{attribute 'linkalways'} 
{attribute 'no_explicit_call' := 'This FB is a CLASS and must be accessed using methods or properties'}
{attribute 'enable_dynamic_creation'}
FUNCTION_BLOCK JsonDeserializer EXTENDS Disposable IMPLEMENTS I_Deserializer
VAR
	jsonParser : JsonDomParser;
	root : SJsonValue;
	garbageCollector : DeserializerGarbageCollector;
	nullNode : JsonDeserializerNullNode;
	rootNode : I_Deserializer := nullNode;
END_VAR

METHOD PUBLIC Clone : I_Deserializer
VAR
	pClone : POINTER TO JsonDeserializer;
	jsonSize : UDINT;
	pJsonString : POINTER TO STRING;
END_VAR
pClone := __NEW(JsonDeserializer);
Clone := pClone^;

jsonSize := jsonParser.GetDocumentLength();

IF jsonSize = 0 THEN
	// no further cloning to do. 
	RETURN;
END_IF

pJsonString := __NEW(BYTE, jsonSize);

IF jsonParser.CopyDocument(pJsonString^, jsonSize) = 0 THEN
	__DELETE(pJsonString);
	RETURN;
END_IF

pClone^.TryLoad(pJsonString^);
__DELETE(pJsonString);
END_METHOD

METHOD PROTECTED CreateDeserializer : I_Deserializer
VAR_INPUT
	DeserializerRoot : SJsonValue;
END_VAR
VAR 
	pNode : POINTER TO JsonDeserializerNode;
END_VAR
pNode := __NEW(JsonDeserializerNode(ParentJsonDomParser := jsonParser, NodeRoot := DeserializerRoot, ParentGarbageCollector := garbageCollector, ParentNullDeserializer := nullNode));
CreateDeserializer := pNode^;
END_METHOD

METHOD FB_exit : BOOL
VAR_INPUT
	bInCopyCode : BOOL; // if TRUE, the exit method is called for exiting an instance that is copied afterwards (online change).
END_VAR
IF bInCopyCode THEN
	RETURN;
END_IF

Reset();
END_METHOD

METHOD GetArray : I_Deserializer
VAR_INPUT
END_VAR
GetArray := rootNode.GetArray();
END_METHOD

METHOD GetElementByIndex : I_Deserializer
VAR_INPUT
	Index : UDINT;
END_VAR
GetElementByIndex := rootNode.GetElementByIndex(Index);
END_METHOD

METHOD GetKey : I_Deserializer
VAR_INPUT
	Key : T_MAXSTRING;
END_VAR
GetKey := rootNode.GetKey(Key);
END_METHOD

METHOD GetKeyArray : I_Deserializer
VAR_INPUT
	Key : T_MAXSTRING;
END_VAR
GetKeyArray := rootNode.GetKeyArray(Key);
END_METHOD

METHOD PUBLIC Reset
VAR_INPUT
END_VAR
jsonParser.NewDocument();
garbageCollector.Execute();
root := 0;
rootNode := nullNode;
END_METHOD

METHOD TryGetBase64 : BOOL
VAR_INPUT
	pBytes : POINTER TO BYTE;
	nBytes : DINT;
END_VAR
TryGetBase64 := rootNode.TryGetBase64(pBytes, nBytes);
END_METHOD

METHOD TryGetBool : BOOL
VAR_INPUT
	Destination : REFERENCE TO BOOL;
END_VAR
TryGetBool := rootNode.TryGetBool(Destination);
END_METHOD

METHOD TryGetByte : BOOL
VAR_INPUT
	Destination : REFERENCE TO BYTE;
END_VAR
TryGetByte := rootNode.TryGetByte(Destination);
END_METHOD

METHOD TryGetDateTime : BOOL
VAR_INPUT
	Destination : REFERENCE TO DATE_AND_TIME;
END_VAR
TryGetDateTime := rootNode.TryGetDateTime(Destination);
END_METHOD

METHOD TryGetDcTime : BOOL
VAR_INPUT
	Destination : REFERENCE TO DCTIME;
END_VAR
TryGetDcTime := rootNode.TryGetDcTime(Destination);
END_METHOD

METHOD TryGetDint : BOOL
VAR_INPUT
	Destination : REFERENCE TO DINT;
END_VAR
TryGetDint := rootNode.TryGetDint(Destination);
END_METHOD

METHOD TryGetDword : BOOL
VAR_INPUT
	Destination : REFERENCE TO DWORD;
END_VAR
TryGetDword := rootNode.TryGetDword(Destination);
END_METHOD

METHOD TryGetFileTime : BOOL
VAR_INPUT
	Destination : REFERENCE TO FILETIME;
END_VAR
TryGetFileTime := rootNode.TryGetFileTime(Destination);
END_METHOD

METHOD TryGetHexAsBytes : BOOL
VAR_INPUT
	pBytes : POINTER TO BYTE;
	nBytes : DINT;
END_VAR
TryGetHexAsBytes := rootNode.TryGetHexAsBytes(pBytes, nBytes);
END_METHOD

METHOD TryGetInt : BOOL
VAR_INPUT
	Destination : REFERENCE TO INT;
END_VAR
TryGetInt := rootNode.TryGetInt(Destination);
END_METHOD

METHOD TryGetKeyBase64 : BOOL
VAR_INPUT
	Key : T_MAXSTRING;
	pBytes : POINTER TO BYTE;
	nBytes : DINT;
END_VAR
TryGetKeyBase64 := rootNode.TryGetKeyBase64(Key, pBytes, nBytes);
END_METHOD

METHOD TryGetKeyBool : BOOL
VAR_INPUT
	Key : T_MAXSTRING;
	Destination : REFERENCE TO BOOL;
END_VAR
TryGetKeyBool := rootNode.TryGetKeyBool(Key, Destination);
END_METHOD

METHOD TryGetKeyByte : BOOL
VAR_INPUT
	Key : T_MAXSTRING;
	Destination : REFERENCE TO BYTE;
END_VAR
TryGetKeyByte := rootNode.TryGetKeyByte(Key, Destination);
END_METHOD

METHOD TryGetKeyDateTime : BOOL
VAR_INPUT
	Key : T_MAXSTRING;
	Destination : REFERENCE TO DATE_AND_TIME;
END_VAR
TryGetKeyDateTime := rootNode.TryGetKeyDateTime(Key, Destination);
END_METHOD

METHOD TryGetKeyDcTime : BOOL
VAR_INPUT
	Key : T_MAXSTRING;
	Destination : REFERENCE TO DCTIME;
END_VAR
TryGetKeyDcTime := rootNode.TryGetKeyDcTime(Key, Destination);
END_METHOD

METHOD TryGetKeyDint : BOOL
VAR_INPUT
	Key : T_MAXSTRING;
	Destination : REFERENCE TO DINT;
END_VAR
TryGetKeyDint := rootNode.TryGetKeyDint(Key, Destination);
END_METHOD

METHOD TryGetKeyDword : BOOL
VAR_INPUT
	Key : T_MAXSTRING;
	Destination : REFERENCE TO DWORD;
END_VAR
TryGetKeyDword := rootNode.TryGetKeyDword(Key, Destination);
END_METHOD

METHOD TryGetKeyFileTime : BOOL
VAR_INPUT
	Key : T_MAXSTRING;
	Destination : REFERENCE TO FILETIME;
END_VAR
TryGetKeyFileTime := rootNode.TryGetKeyFileTime(Key, Destination);
END_METHOD

METHOD TryGetKeyHexAsBytes : BOOL
VAR_INPUT
	Key : T_MAXSTRING;
	pBytes : POINTER TO BYTE;
	nBytes : DINT;
END_VAR
TryGetKeyHexAsBytes := rootNode.TryGetKeyHexAsBytes(Key, pBytes, nBytes);
END_METHOD

METHOD TryGetKeyInt : BOOL
VAR_INPUT
	Key : T_MAXSTRING;
	Destination : REFERENCE TO INT;
END_VAR
TryGetKeyInt := rootNode.TryGetKeyInt(Key, Destination);
END_METHOD

METHOD TryGetKeyLint : BOOL
VAR_INPUT
	Key : T_MAXSTRING;
	Destination : REFERENCE TO LINT;
END_VAR
TryGetKeyLint := rootNode.TryGetKeyLint(Key, Destination);
END_METHOD

METHOD TryGetKeyLreal : BOOL
VAR_INPUT
	Key : T_MAXSTRING;
	Destination : REFERENCE TO LREAL;
END_VAR
TryGetKeyLreal := rootNode.TryGetKeyLreal(Key, Destination);
END_METHOD

METHOD TryGetKeyLtime : BOOL
VAR_INPUT
	Key : T_MAXSTRING;
	Destination : REFERENCE TO LTIME;
END_VAR
TryGetKeyLtime := rootNode.TryGetKeyLtime(Key, Destination);
END_METHOD

METHOD TryGetKeyLword : BOOL
VAR_INPUT
	Key : T_MAXSTRING;
	Destination : REFERENCE TO LWORD;
END_VAR
TryGetKeyLword := rootNode.TryGetKeyLword(Key, Destination);
END_METHOD

METHOD TryGetKeyObject : BOOL
VAR_INPUT
	Key : T_MAXSTRING;
	Object : I_Deserializable;
END_VAR
TryGetKeyObject := rootNode.TryGetKeyObject(Key,Object);
END_METHOD

METHOD TryGetKeyReal : BOOL
VAR_INPUT
	Key : T_MAXSTRING;
	Destination : REFERENCE TO REAL;
END_VAR
TryGetKeyReal := rootNode.TryGetKeyReal(Key, Destination);
END_METHOD

METHOD TryGetKeySint : BOOL
VAR_INPUT
	Key : T_MAXSTRING;
	Destination : REFERENCE TO SINT;
END_VAR
TryGetKeySint := rootNode.TryGetKeySint(Key, Destination);
END_METHOD

METHOD TryGetKeyString : BOOL
VAR_INPUT
	Key : T_MAXSTRING;
	Destination : REFERENCE TO STRING;
END_VAR
TryGetKeyString := rootNode.TryGetKeyString(Key, Destination);
END_METHOD

METHOD TryGetKeyTime : BOOL
VAR_INPUT
	Key : T_MAXSTRING;
	Destination : REFERENCE TO TIME;
END_VAR
TryGetKeyTime := rootNode.TryGetKeyTime(Key, Destination);
END_METHOD

METHOD TryGetKeyTod : BOOL
VAR_INPUT
	Key : T_MAXSTRING;
	Destination : REFERENCE TO TOD;
END_VAR
TryGetKeyTod := rootNode.TryGetKeyTod(Key, Destination);
END_METHOD

METHOD TryGetKeyUdint : BOOL
VAR_INPUT
	Key : T_MAXSTRING;
	Destination : REFERENCE TO UDINT;
END_VAR
TryGetKeyUdint := rootNode.TryGetKeyUdint(Key, Destination);
END_METHOD

METHOD TryGetKeyUint : BOOL
VAR_INPUT
	Key : T_MAXSTRING;
	Destination : REFERENCE TO UINT;
END_VAR
TryGetKeyUint := rootNode.TryGetKeyUint(Key, Destination);
END_METHOD

METHOD TryGetKeyUlint : BOOL
VAR_INPUT
	Key : T_MAXSTRING;
	Destination : REFERENCE TO ULINT;
END_VAR
TryGetKeyUlint := rootNode.TryGetKeyUlint(Key, Destination);
END_METHOD

METHOD TryGetKeyUsint : BOOL
VAR_INPUT
	Key : T_MAXSTRING;
	Destination : REFERENCE TO USINT;
END_VAR
TryGetKeyUsint := rootNode.TryGetKeyUsint(Key, Destination);
END_METHOD

METHOD TryGetKeyWord : BOOL
VAR_INPUT
	Key : T_MAXSTRING;
	Destination : REFERENCE TO WORD;
END_VAR
TryGetKeyWord := rootNode.TryGetKeyWord(Key, Destination);
END_METHOD

METHOD TryGetLint : BOOL
VAR_INPUT
	Destination : REFERENCE TO LINT;
END_VAR
TryGetLint := rootNode.TryGetLint(Destination);
END_METHOD

METHOD TryGetLreal : BOOL
VAR_INPUT
	Destination : REFERENCE TO LREAL;
END_VAR
TryGetLreal := rootNode.TryGetLreal(Destination);
END_METHOD

METHOD TryGetLtime : BOOL
VAR_INPUT
	Destination : REFERENCE TO LTIME;
END_VAR
TryGetLtime := rootNode.TryGetLtime(Destination);
END_METHOD

METHOD TryGetLword : BOOL
VAR_INPUT
	Destination : REFERENCE TO LWORD;
END_VAR
TryGetLword := rootNode.TryGetLword(Destination);
END_METHOD

METHOD TryGetObject : BOOL
VAR_INPUT
	Object : I_Deserializable;
END_VAR
TryGetObject := rootNode.TryGetObject(Object);
END_METHOD

METHOD TryGetReal : BOOL
VAR_INPUT
	Destination : REFERENCE TO REAL;
END_VAR
TryGetReal := rootNode.TryGetReal(Destination);
END_METHOD

METHOD TryGetSint : BOOL
VAR_INPUT
	Destination : REFERENCE TO SINT;
END_VAR
TryGetSint := rootNode.TryGetSint(Destination);
END_METHOD

METHOD TryGetString : BOOL
VAR_INPUT
	Destination : REFERENCE TO STRING;
END_VAR
TryGetString := rootNode.TryGetString(Destination);
END_METHOD

METHOD TryGetTime : BOOL
VAR_INPUT
	Destination : REFERENCE TO TIME;
END_VAR
TryGetTime := rootNode.TryGetTime(Destination);
END_METHOD

METHOD TryGetTod : BOOL
VAR_INPUT
	Destination : REFERENCE TO TOD;
END_VAR
TryGetTod := rootNode.TryGetTod(Destination);
END_METHOD

METHOD TryGetUdint : BOOL
VAR_INPUT
	Destination : REFERENCE TO UDINT;
END_VAR
TryGetUdint := rootNode.TryGetUdint(Destination);
END_METHOD

METHOD TryGetUint : BOOL
VAR_INPUT
	Destination : REFERENCE TO UINT;
END_VAR
TryGetUint := rootNode.TryGetUint(Destination);
END_METHOD

METHOD TryGetUlint : BOOL
VAR_INPUT
	Destination : REFERENCE TO ULINT;
END_VAR
TryGetUlint := rootNode.TryGetUlint(Destination);
END_METHOD

METHOD TryGetUsint : BOOL
VAR_INPUT
	Destination : REFERENCE TO USINT;
END_VAR
TryGetUsint := rootNode.TryGetUsint(Destination);
END_METHOD

METHOD TryGetWord : BOOL
VAR_INPUT
	Destination : REFERENCE TO WORD;
END_VAR
TryGetWord := rootNode.TryGetWord(Destination);
END_METHOD

METHOD PUBLIC TryLoad : BOOL
VAR_INPUT
	SerializedData : REFERENCE TO STRING;;
END_VAR
Reset();

root := jsonParser.ParseDocument(SerializedData);
IF root = 0 THEN
	RETURN;
END_IF

rootNode := CreateDeserializer(root);
TryLoad := TRUE;
END_METHOD

END_FUNCTION_BLOCK

(* stored: Version 1.1.0.1, ProductVersion 3.1.4024.12
   POU JsonDeserializer: Id {a90a43d9-ea62-48ae-9b56-2bc4217891a9}, SpecialFunc None
   Folder Destructor: Id {bf822394-22a2-42d6-8812-78eace02343d}
   Folder Protected: Id {01c55fae-a423-471f-adbb-267168f4fce0}
   Method Clone: Id {f09ba639-152e-42ab-83f4-0db39532c374}
   Method CreateDeserializer: Id {6e178c51-cb69-40a4-96bf-b38252df7bdc}
   Method FB_exit: Id {d9f286cf-0a82-45b5-9661-1cb5706a832d}
   Method GetArray: Id {a8b524f2-5f76-4824-97b5-f83f0e1611cd}
   Method GetElementByIndex: Id {adfb94ab-88ff-476c-a549-f0880b6a7e45}
   Method GetKey: Id {0f1075b2-7f5b-4f71-8323-87a91a30b569}
   Method GetKeyArray: Id {64ed3b17-47ab-402e-a2fe-0b75f40cb73a}
   Method Reset: Id {ff410b24-6bd3-4b0b-b181-8baf610127fb}
   Method TryGetBase64: Id {fe295ea1-6385-4c90-8c1e-0130d0abea78}
   Method TryGetBool: Id {6ec60297-fc78-4e42-8c9b-b797b172a63d}
   Method TryGetByte: Id {7f56b251-eee0-4e1f-94af-df45fa90da48}
   Method TryGetDateTime: Id {0eefca34-6e86-480c-bd80-cca9f9d6217f}
   Method TryGetDcTime: Id {822c1511-2a5b-4b36-a7ac-0e7bb0382e3f}
   Method TryGetDint: Id {72d1a2f6-6d1c-43bc-8260-7a62f2ef0180}
   Method TryGetDword: Id {92993be7-2fb3-49bb-aa8c-994491f8b23c}
   Method TryGetFileTime: Id {6f985b02-908a-4e9a-8047-f818f837fe22}
   Method TryGetHexAsBytes: Id {57725d6f-7769-44f1-b87a-65ec295b3672}
   Method TryGetInt: Id {2fdf166b-5700-40ee-b8b0-abadc2efc46c}
   Method TryGetKeyBase64: Id {e2e97d9b-41bc-414a-9d61-b71ea3e26097}
   Method TryGetKeyBool: Id {5f267a8c-ebc4-4c51-b0f0-4a95026c8a3f}
   Method TryGetKeyByte: Id {1c43e54c-ee47-4d7b-bcae-5f660a8fcad5}
   Method TryGetKeyDateTime: Id {c22b8398-2c86-4d72-9120-e789b40c9718}
   Method TryGetKeyDcTime: Id {38227bfb-4cf2-495f-acbb-91f5f470f11e}
   Method TryGetKeyDint: Id {82fdf3a0-94c2-4a8e-923d-cf45ec507d72}
   Method TryGetKeyDword: Id {5a45d2b3-e2ba-457e-a3e4-d79c9082fa74}
   Method TryGetKeyFileTime: Id {ce1ac8be-a887-4bce-96e2-9b3a4179a8cb}
   Method TryGetKeyHexAsBytes: Id {6d3a64ed-e904-4405-97e8-629172119dae}
   Method TryGetKeyInt: Id {9d78e31a-c0cd-4dc2-a6c9-cc7bb2a5aeb5}
   Method TryGetKeyLint: Id {d12995f5-5579-4299-9a40-19fd2107eff5}
   Method TryGetKeyLreal: Id {92c3eaf3-71df-4e2f-ba93-315676c41524}
   Method TryGetKeyLtime: Id {f0eafc1e-bf4b-4ceb-bdeb-6ae313a3df89}
   Method TryGetKeyLword: Id {65ebf9c9-8746-4bf0-9897-02e88608bc54}
   Method TryGetKeyObject: Id {62ed7c8c-f671-47eb-b767-f4d091a68ae9}
   Method TryGetKeyReal: Id {ba9c869b-cf53-471e-bda6-414ea929fcfa}
   Method TryGetKeySint: Id {9c210d46-b2cf-4e87-b34c-9c31c974981c}
   Method TryGetKeyString: Id {145e945a-6148-465d-8d1e-78bff0346911}
   Method TryGetKeyTime: Id {ac1c2336-2654-4ecb-9c0d-cdf530414a88}
   Method TryGetKeyTod: Id {bde0ce6f-cd97-4fe6-9b33-f96250f01eed}
   Method TryGetKeyUdint: Id {3f71ab6a-2c21-48ba-bea8-ac9c531c6a2f}
   Method TryGetKeyUint: Id {b09d8575-090d-49e4-a0ce-27fe71c91a45}
   Method TryGetKeyUlint: Id {499ee358-c7a9-4f43-9581-abd422c87ec8}
   Method TryGetKeyUsint: Id {35f67b71-f2b8-4d86-9bb3-95ee1284ba30}
   Method TryGetKeyWord: Id {7efab29f-f53c-471a-95c5-75e9be77a68f}
   Method TryGetLint: Id {75731b5e-e042-400b-a3d1-9b9ba60506d8}
   Method TryGetLreal: Id {7b380507-57f2-4a93-985b-86be64078e31}
   Method TryGetLtime: Id {efd7f5a3-8843-4642-bc86-b9940affcca4}
   Method TryGetLword: Id {0295afb4-f050-4895-9c0b-6b9cdfa8b1ee}
   Method TryGetObject: Id {4a3bb941-939c-4dd6-bed5-5312803ff942}
   Method TryGetReal: Id {6c3290d3-fec4-47f7-a5d0-1861de90ccaf}
   Method TryGetSint: Id {e84565ff-7164-409c-9f95-c7b2be3fbcff}
   Method TryGetString: Id {44240e6f-9963-4706-910b-e5c87c3f8607}
   Method TryGetTime: Id {80d80d87-f037-436c-8f8f-7f8fec352f39}
   Method TryGetTod: Id {9e042969-ff4a-4b34-89ea-b8144dd0d5ca}
   Method TryGetUdint: Id {751bec7e-3a00-432c-b241-6a6fad2970fb}
   Method TryGetUint: Id {972566ca-529a-4fb3-bb50-96a823c8709e}
   Method TryGetUlint: Id {3f4a2c33-9649-45c1-875c-327dc26bc3a5}
   Method TryGetUsint: Id {17108ee2-2a2f-480d-a20a-5a3943e8a7ad}
   Method TryGetWord: Id {39e3134f-9f16-4677-84f1-71254c101d0e}
   Method TryLoad: Id {f075a62d-029d-4d3a-a33f-32a6021b89c2} *)
